Staubli VAL3: F6_DELT.pgx

program F6_DELT()
begin
  while size(sString)>1
    $ddel(sString,size(sString)-1)
  endWhile
  while size(pfrmCad)>1
    $ddel(pfrmCad,size(pfrmCad)-1)
  endWhile
  while size(nPulse)>1
    $ddel(nPulse,size(nPulse)-1)
  endWhile
  n_sTxt=0
  sScrPts="NotReady"
  call hmi_refreshmain()
  popUpMsg("数据已清空,可以关机")

end
